# EPICS autosave request: autosave/galil_profileMoveController.req
$(P)$(R):TrajectoryFile
$(P)$(R):PROFILETYPE_CMD
